// Mitsubishi GX Works2 project: 타이머실습0   PLC: Q03UDV

PROGRAM MAIN
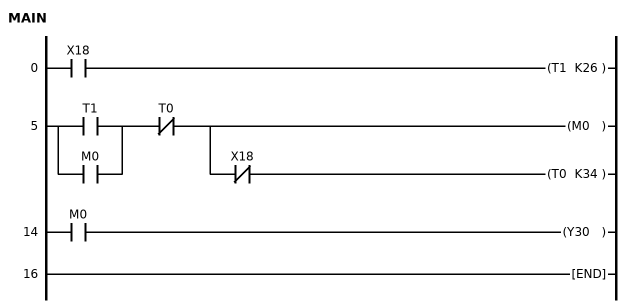
0     LD      X18
      OUT     T1 K26
5     LD      T1
      OR      M0
      ANI     T0
      OUT     M0
      ANI     X18
      OUT     T0 K34
14    LD      M0
      OUT     Y30
16    END
END_PROGRAM
